// SIMATIC S7-200 project (STEP 7-Micro/WIN), CPU 224 REL 01.10

ORGANIZATION_BLOCK MAIN:OB1
TITLE=系统允许操作员通过时间设定标志设定PLC的系统时间：当时间设定标志置为1时，系统将预设的年、月、日、时、分、秒、星期（均为BCD码格式）写入对应地址。在时间设定标志的上升沿，系统通过TODW指令将这些数据写入PLC时钟，完成时间更新——此操作仅在上升沿执行，避免重复写入导致时间错误。设定完成后，操作员需手动复位时间设定标志，以防止持续置位引发重复操作。
// 与此同时，系统通过始终接通标志持续驱动时间读取任务：周期性执行TODR指令，从PLC时钟读取当前时间并存入时间读取存储。随后，系统将时间读取存储中的BCD码数据逐字节转换为整数格式，分别存入年份显示存储、月份显示存储、日期显示存储、小时显示存储、分钟显示存储、秒钟显示存储和星期显示存储。这一转换过程通过BTI指令完成，确保从BCD码到整数的准确性；转换在时间读取后由始终接通标志驱动执行，以保证显示时间的实时更新。通过这样的设计，系统为化工厂提供了一个可靠的时间管理模块，确保生产流程的时间协调。
BEGIN
Network 1 // 将当前时间设定到S7-200当中 ----> VB100:年  VB101:月  VB102:日  VB103:时  VB104:秒  VB107:星期   
// 将当前时间移动到VB100--VB107
LD     M0.0
MOVB   16#3, VB100
MOVB   16#9, VB101
MOVB   16#11, VB102
MOVB   16#9, VB103
MOVB   16#30, VB104
MOVB   16#0, VB105
MOVB   16#0, VB106
MOVB   16#4, VB107
Network 2 // 通过M0.0的一个上升沿将上一步设定的时间写入到S7-200的时钟当中。
// 当M0.0出现一次上升沿，将上面所设定的时间写入到PLC当中
LD     M0.0
EU
TODW   VB100
Network 3 // 设定时间后，可以通过这句话实时读取PLC当中的时间
// 从PLC中读出当前的时间
LD     SM0.0
TODR   VB110
Network 4 // 将读到的结果从BCD码格式转换到整数格式。
----> VW200:年  VW202:月  VB102:日  VB103:时  VB104:秒  VB107:星期  
// 将当前时间移动到VB100--VB107
LD     SM0.0
LPS
BTI    VB110, VW200
AENO
BCDI   VW200
LRD
BTI    VB111, VW202
AENO
BCDI   VW202
LRD
BTI    VB112, VW204
AENO
BCDI   VW204
LRD
BTI    VB113, VW206
AENO
BCDI   VW206
LRD
BTI    VB114, VW208
AENO
BCDI   VW208
LRD
BTI    VB115, VW210
AENO
BCDI   VW210
LRD
BTI    VB116, VW212
AENO
BCDI   VW212
LPP
BTI    VB117, VW214
AENO
BCDI   VW214
END_ORGANIZATION_BLOCK
